TYPE ST_Alarm :
STRUCT
    nID : UINT;
    eSeverity : E_AlarmSeverity;
    eState : E_AlarmState;
    sMessage : STRING(80);
    sSource : STRING(40);
    tRaiseTime : DT;
    tAckTime : DT;
    tClearTime : DT;
    bRequiresAck : BOOL;
    bSelfClearing : BOOL;
END_STRUCT
END_TYPE

(* stored: Version 1.1.0.1
   DUT ST_Alarm: Id {8C84B5D4-45BD-3AFF-6E09-1CCBA7C6AD54} *)
